RoboDK station: INSPECCION.rdk

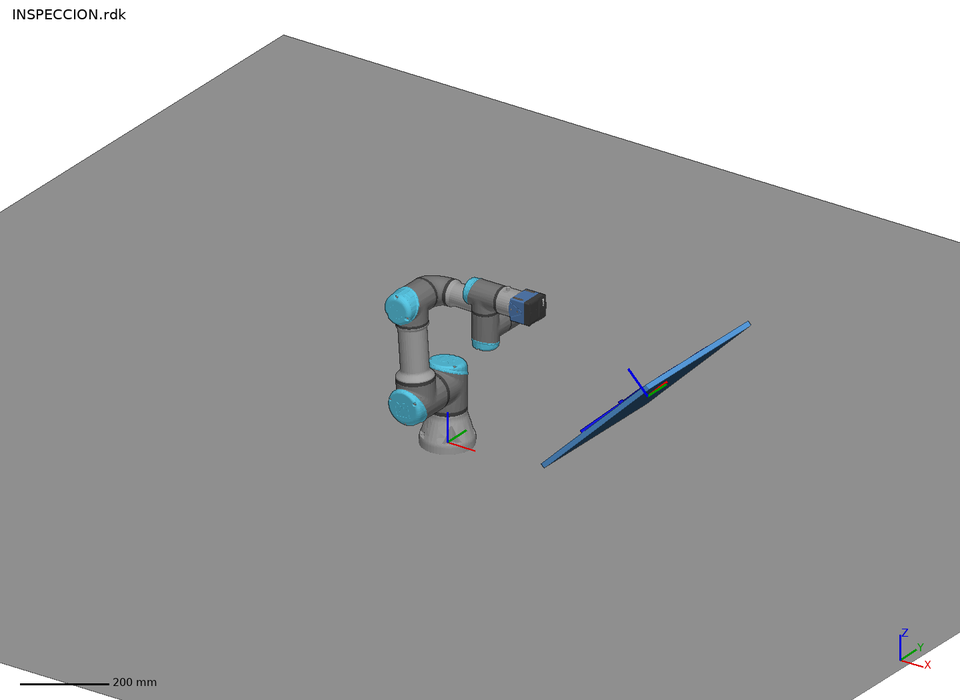
[picture v0: the station drawn from its stored meshes, robots at their saved joint values, targets as dots, program paths as lines]
Station INSPECCION (saved by RoboDK 5.7.3). Poses are relative to the parent item; angles as X-Y-Z fixed-axis rotations.
  - frame UR3e Base at (0, 0, 0) mm
    - robot UR3e: 6 axes, payload 3 kg, reach 500 mm, repeatability 0.03 mm, weight 11 kg
        modified DH rows (alpha deg, a mm, theta deg, d mm): 0, 0, 0, 151.9; 90, 0, 180, 0; 0, 243.55, 0, 0; 0, 213.2, 0, 131.05; -90, 0, 0, 85.35; 90, 0, 180, 92.1
        joint limits [-360, -360, -360, -360, -360, -360] to [360, 360, 360, 360, 360, 360]; home [0, -90, -90, 0, 90, 0]; saved at [0, -85.937, -94.819, 0.756, 90, 0]
      - tool SICK PLB540 Camera, TCP at (0, 0, 160) mm, size 64 x 56 x 62 mm, geometry from SICK-PLB540-Camera.sld
  - frame Frame 2 at (570.77, -31.54, 286.83) mm, rotated rx 0 ry -44 rz 0 deg
    - object RoboDK RDK Plate 100x100mm at (0, 0, 0) mm, rotated rx 0 ry 0 rz 180 deg, size 400 x 400 x 20 mm, geometry from RoboDK-RDK-Plate-100x100mm.sld
  - frame Frame 3 at (0, 0, 0) mm
    - object Floor at (0, 0, 0) mm, size 3000 x 3000 x 0 mm, geometry from Floor.sld
